(* Schneider Machine Expert - Basic project Run Hour2, file version 1.7.0.0 *)
(* ProjectInformations: Name=New project *)

HARDWARE
  Cpu 0: TM221ME32TK
  EthernetConfiguration: NetworkName=M221, IpAllocationMode=FixedAddress, IpAddress=0.0.0.0, SubnetMask=0.0.0.0
  SerialLineConfiguration: Baud=Baud19200, Parity=ParityEven, DataBits=DataBits8, StopBits=StopBits1, PhysicalMedium=PhysicalMediumRs485, TransmissionMode=TransmissionModeModbusRtu, SlaveId=1, Addressing=SlaveAddressing
  MastTask: UsePeriodScanMode=false, PeriodScan=100
  FastTask: Period=255
  CpuBehavior: StartingMode=StartAsPreviousState, AutoSaveRamOnEeprom=true, WatchdogPeriod=250

SYMBOLS  (address, symbol, comment, settings)
  %TM1        "T1"  [Preset=6, Base=OneSecond]
  %TM2        "T2"  [Preset=6, Base=OneSecond]
  %TM3        [Preset=1, Base=OneSecond, IsRetentive=true]
  %TM4        [Preset=1, Base=OneSecond, IsRetentive=true]
  %I0.0       "Auto"
  %I0.1       "Manual"
  %I0.2       "Pompa 1"
  %I0.3       "Pompa 2"
  %Q0.0       "P1"
  %Q0.1       "P2"

POU New POU
  (* SectionNumber=1 *)

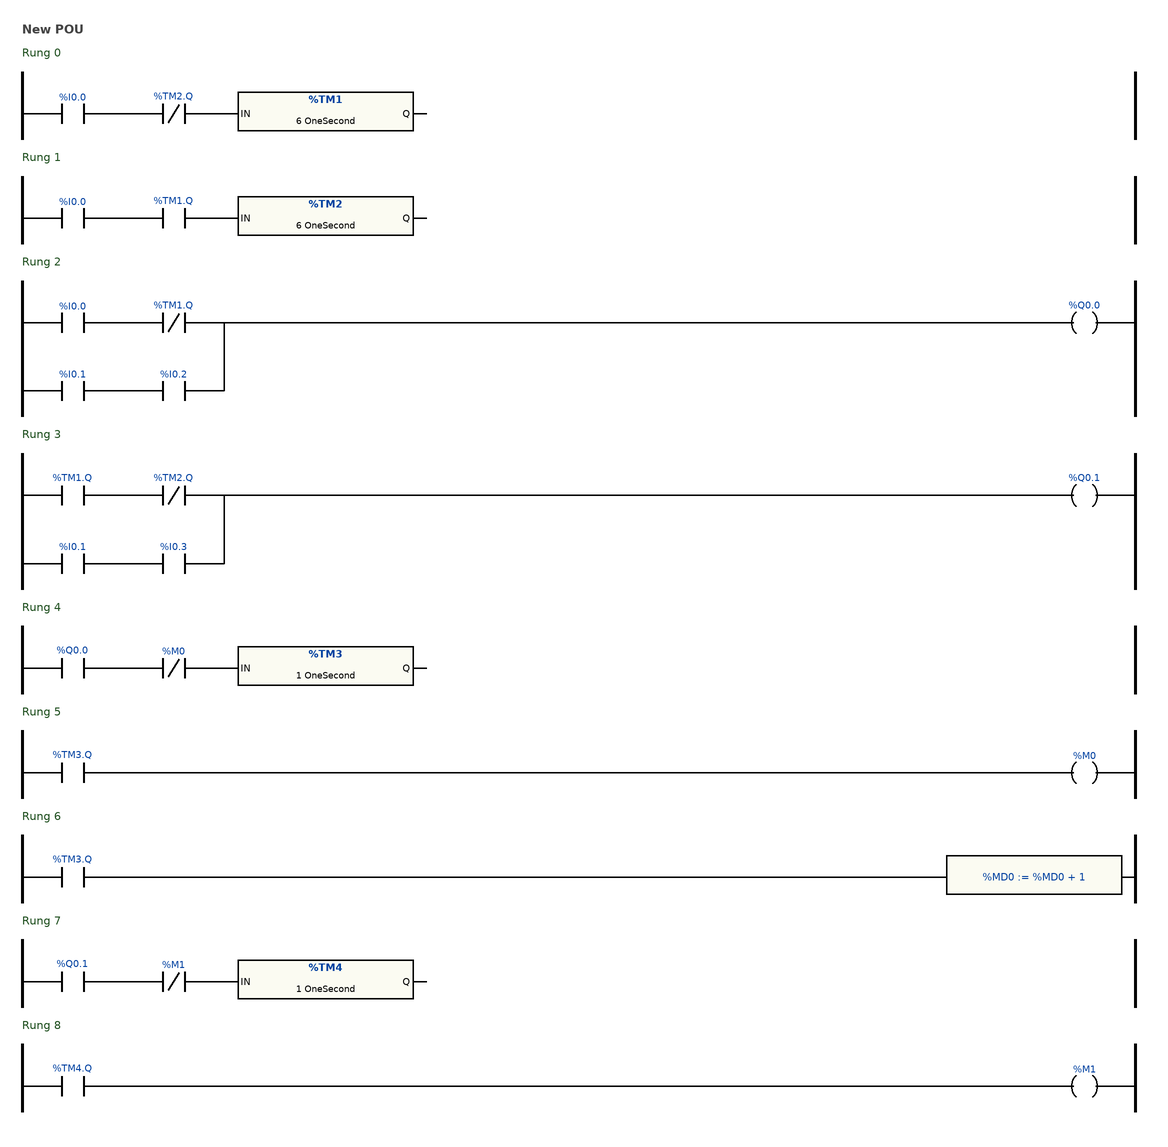

// Rung 0
  BLK %TM1
  LD %I0.0
  ANDN %TM2.Q
  IN
  END_BLK
  // as ST:
  //   %TM1(IN := %I0.0 AND NOT %TM2.Q);

// Rung 1
  BLK %TM2
  LD %I0.0
  AND %TM1.Q
  IN
  END_BLK
  // as ST:
  //   %TM2(IN := %I0.0 AND %TM1.Q);

// Rung 2
  LD %I0.0
  ANDN %TM1.Q
  OR( %I0.1
  AND %I0.2
  )
  ST %Q0.0
  // as ST:
  //   %Q0.0 := %I0.0 AND NOT %TM1.Q OR %I0.1 AND %I0.2;

// Rung 3
  LD %TM1.Q
  ANDN %TM2.Q
  OR( %I0.1
  AND %I0.3
  )
  ST %Q0.1
  // as ST:
  //   %Q0.1 := %TM1.Q AND NOT %TM2.Q OR %I0.1 AND %I0.3;

// Rung 4
  BLK %TM3
  LD %Q0.0
  ANDN %M0
  IN
  END_BLK
  // as ST:
  //   %TM3(IN := %Q0.0 AND NOT %M0);

// Rung 5
  LD %TM3.Q
  ST %M0
  // as ST:
  //   %M0 := %TM3.Q;

// Rung 6
  LD %TM3.Q
  [ %MD0 := %MD0 + 1 ]
  // as ST:
  //   IF %TM3.Q THEN %MD0 := %MD0 + 1; END_IF;

// Rung 7
  BLK %TM4
  LD %Q0.1
  ANDN %M1
  IN
  END_BLK
  // as ST:
  //   %TM4(IN := %Q0.1 AND NOT %M1);

// Rung 8
  LD %TM4.Q
  ST %M1
  // as ST:
  //   %M1 := %TM4.Q;

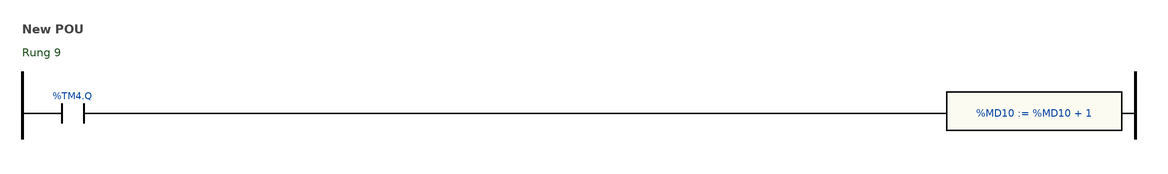

// Rung 9
  LD %TM4.Q
  [ %MD10 := %MD10 + 1 ]
  // as ST:
  //   IF %TM4.Q THEN %MD10 := %MD10 + 1; END_IF;
